FUNCTION_BLOCK FB_BagCompactor
VAR_INPUT
  ams_net_id: STRING;
END_VAR
VAR_OUTPUT
END_VAR
VAR
  status: BagMachineStatus;
  error_code: UINT;
END_VAR

{attribute 'TcRpcEnable'}
METHOD PUBLIC compact_bag : BOOL
VAR_INPUT

END_VAR
END_METHOD

END_FUNCTION_BLOCK

(* stored: Version 1.1.0.1, ProductVersion 3.1.4024.12
   POU FB_BagCompactor: Id {017b6eb5-a8fd-4f32-9753-e8dab8e3fb07}, SpecialFunc None
   Method compact_bag: Id {d356716c-e9b9-41b0-91db-30267c691488} *)
